Staubli VAL3: Str_SplitComma.pgx

program Str_SplitComma(bool& x_bRes, string x_sStrIn, string& x_sOut[])
begin
  //****************************************************************
  //***************************************************************
  //函数名称：SplitChar
  //用途：  用于解析字符
  //创建日期：
  //作者：
  //联系方式：
  //备注：传入的数组个数决定了其中的分配
  //版本修改说明：
  //****************************************************************
  //*****************************************************************
  call Str_SplitChar(x_bRes,x_sStrIn,",",x_sOut)
end
